TYPE ST_PrefireDiscon_Base :
STRUCT
	PrefireDisconClosed			: BOOL := FALSE;
	PrefireDisconOpen			: BOOL := FALSE;
	ChargePrefireDisconCap		: BOOL := FALSE;   //1 = charge, 0 = dump?
	ClosePrefireDiscon			: BOOL := FALSE;
END_STRUCT
END_TYPE

(* stored: Version 1.1.0.1, ProductVersion 3.1.4024.11
   DUT ST_PrefireDiscon_Base: Id {1a40a9e0-e046-4d70-885d-502a970c6eab} *)
